PROGRAM GEMMA
VAR
	STEP_A6: INT := 0;
	DELAY_EJECTION_CARRIERS: TON;
	EJECT_CARRIERS: BOOL;
	F2_END: BOOL;
	STEP: STRING(20);
END_VAR

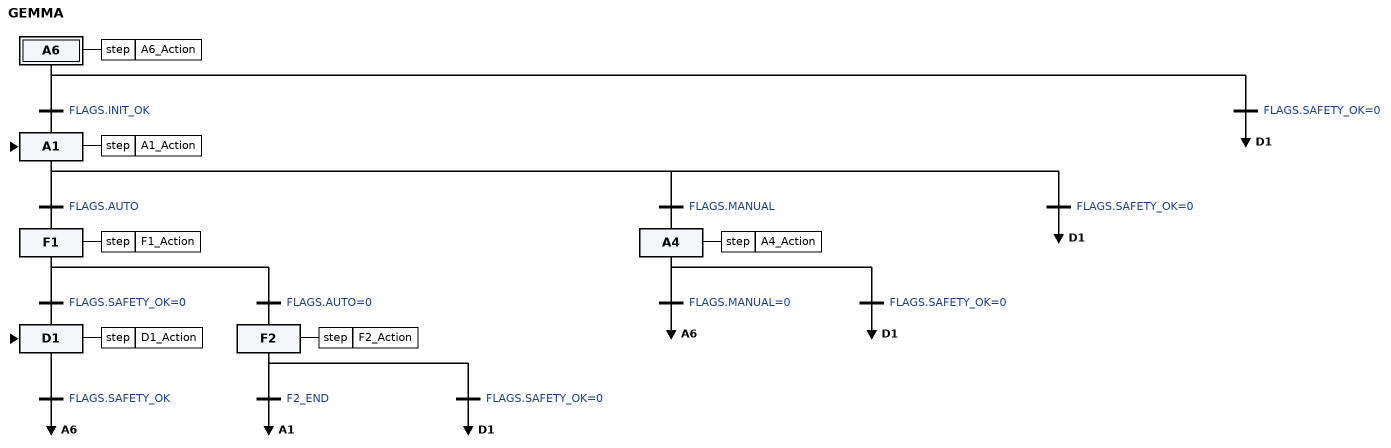
INITIAL_STEP A6_:  // name as stored: A6 
    A6_Action(N);  // step action
END_STEP
TRANSITION FROM A6_ TO A1
    := FLAGS.INIT_OK;
END_TRANSITION
TRANSITION FROM A6_ TO D1
    := FLAGS.SAFETY_OK=0;
END_TRANSITION
STEP A1:
    A1_Action(N);  // step action
END_STEP
TRANSITION FROM A1 TO F1
    := FLAGS.AUTO;
END_TRANSITION
TRANSITION FROM A1 TO A4
    := FLAGS.MANUAL;
END_TRANSITION
STEP A4:
    A4_Action(N);  // step action
END_STEP
TRANSITION FROM A4 TO A6
    := FLAGS.MANUAL=0;
END_TRANSITION
TRANSITION FROM A4 TO D1
    := FLAGS.SAFETY_OK=0;
END_TRANSITION
TRANSITION FROM A1 TO D1
    := FLAGS.SAFETY_OK=0;
END_TRANSITION
STEP F1:
    F1_Action(N);  // step action
END_STEP
TRANSITION FROM F1 TO D1
    := FLAGS.SAFETY_OK=0;
END_TRANSITION
TRANSITION FROM F1 TO F2
    := FLAGS.AUTO=0;
END_TRANSITION
STEP F2:
    F2_Action(N);  // step action
END_STEP
TRANSITION FROM F2 TO A1
    := F2_END;
END_TRANSITION
TRANSITION FROM F2 TO D1
    := FLAGS.SAFETY_OK=0;
END_TRANSITION
STEP D1:
    D1_Action(N);  // step action
END_STEP
TRANSITION FROM D1 TO A6
    := FLAGS.SAFETY_OK;
END_TRANSITION

ACTION F1_Action:
(*********************************************************
*
* F1
*
************************************************************)

STEP := 'F1';
END_ACTION

ACTION A6_Action:
(**************************************************************
*
*
* Initialisation
*
*
***************************************************************)
STEP:='A6';



CASE STEP_A6 OF

0: (*Init*)
	STEP_A6:=STEP_A6+1;

1: (*Initialise valves and variables*)

	GEN_1V1 				:=FALSE;	(*Vanne AIR*)
	GEN_CONVOYEUR			:=FALSE;	(*Relais convoyeur*)	
	
	ST1_1V1 	:=FALSE;		(*Vérin palette attente*)
	ST1_1V2 	:=FALSE;		(*Vérin palette bloquage*)
	ST1_1V3 	:=FALSE;		(*Vérin palette stop*)
	ST1_1V4 	:=FALSE;		(*Vérin connexion TOP*)
	ST1_1V5		:=FALSE;		(*Vérin connexion HT*)

	ST2_2V1 	:=FALSE;		(*Vérin palette attente*)
	ST2_2V2 	:=FALSE;		(*Vérin palette bloquage*)
	ST2_2V3 	:=FALSE;		(*Vérin palette stop*)
	ST2_2V4 	:=FALSE;		(*Vérin Hydro TOP*)
	ST2_2V5		:=FALSE;		(*Vérin hydro BOTTOM*)
	ST2_2V6		:=FALSE;		(*Vérin électrique*)
	ST2_2V7		:=FALSE;		(*Vérin by-pass*)
	
	ST2_POWER	:=FALSE;		(*Alimentation électrique pompe*)
	
	ST3_3V1 	:=FALSE;		(*Vérin palette attente*)
	ST3_3V2 	:=FALSE;		(*Vérin palette bloquage*)
	ST3_3V3 	:=FALSE;		(*Vérin palette stop*)
	ST3_3V4 	:=FALSE;		(*Vérin Hydro TOP*)
	ST3_3V5		:=FALSE;		(*Vérin hydro BOTTOM*)
	ST3_3V7		:=FALSE;		(*Vérin by-pass*)
	
	ST3_3V10 	:=FALSE;		(*Vanne avant la pompe*)
	ST3_3V11 	:=FALSE;		(*Vanne après la pompe*)
	ST3_3V12 	:=FALSE;		(*Vanne de blocage d'air pour le DELTA*)
	
	ST4_4V1 	:=FALSE;		(*Vérin palette attente*)
	ST4_4V2 	:=FALSE;		(*Vérin palette bloquage*)
	ST4_4V3 	:=FALSE;		(*Vérin palette stop*)
	ST4_4V4 	:=FALSE;		(*Vérin Hydro TOP*)
	ST4_4V5		:=FALSE;		(*Vérin hydro BOTTOM*)
	ST4_4V6		:=FALSE;		(*Vérin électrique*)
	ST4_4V7		:=FALSE;		(*Vérin by-pass*)
	
	ST4_4V10	:=FALSE;		(*Vanne avant la pompe*)
	ST4_4V12	:=FALSE;		(*Vanne après la vanne pilotée*)
	ST4_4V13	:=FALSE;		(*Vanne max flow*)

	ST4_POWER	:=FALSE;		(*Alimentation électrique pompe*)
	ST4_VIDANGE	:=FALSE;		(*Vidange balance*)
	
	ST5_5V1 	:=FALSE;		(*Vérin palette attente*)
	ST5_5V2 	:=FALSE;		(*Vérin palette bloquage*)
	ST5_5V3 	:=FALSE;		(*Vérin palette stop*)
	ST5_5V4 	:=FALSE;		(*Vérin Hydro TOP*)
	ST5_5V5		:=FALSE;		(*Vérin hydro BOTTOM*)
	ST5_5V6		:=FALSE;		(*Vérin électrique*)
	
	ST5_5V10	:=FALSE;		(*Vanne avant la pompe*)
	ST5_5V12	:=FALSE;		(*Vanne après la vanne pilotée*)
	ST5_5V13	:=FALSE;		(*Vanne max flow*)
	
	ST5_5V14	:=FALSE;		(*Vanne vidange vers égouts ou réservoir*)
	ST5_5V15	:=FALSE;			(*Vanne avant la pompe*)
	ST5_5V16	:=FALSE;		(*Vanne provenance eau du réservoir ou du déminéralisateur*)
	
	ST5_POWER	:=FALSE;		(*Alimentation électrique pompe*)
	ST5_VIDANGE	:=FALSE;		(*Vidange balance*)
	
	ST6_6V1 	:=FALSE;		(*Vérin palette attente*)
	ST6_6V2 	:=FALSE;		(*Vérin palette bloquage*)
	ST6_6V3 	:=FALSE;		(*Vérin palette stop*)
	ST6_6V4 	:=FALSE;		(*Vérin Hydro TOP*)
	ST6_6V5		:=FALSE;		(*Vérin hydro BOTTOM*)
	ST6_6V6		:=FALSE;		(*Vérin électrique*)
	ST6_6V7		:=FALSE;		(*Vérin by-pass*)
	
	ST6_6V10	:=FALSE;		(*Vanne avant la pompe*)
	ST6_6V11	:=FALSE;		(*Vanne après la pompe*)
	
	ST6_POWER	:=FALSE;		(*Alimentation électrique pompe*)
	
	ST7_7V1 	:=FALSE;		(*Vérin palette attente*)
	ST7_7V2 	:=FALSE;		(*Vérin palette bloquage*)
	ST7_7V3 	:=FALSE;		(*Vérin palette stop*)
	ST7_7V4 	:=FALSE;		(*Vérin Hydro TOP*)
	ST7_7V5		:=FALSE;		(*Vérin hydro BOTTOM*)
	ST7_7V6		:=FALSE;		(*Vérin électrique*)
	ST7_7V7		:=FALSE;		(*Vérin by-pass*)
	
	ST7_7V10	:=FALSE;		(*Vanne avant la pompe*)
	
	ST7_POWER	:=FALSE;		(*Alimentation électrique pompe*)
	
	ST8_8V1 	:=FALSE;		(*Vérin palette attente*)
	ST8_8V2 	:=FALSE;		(*Vérin palette bloquage*)
	ST8_8V3 	:=FALSE;		(*Vérin palette stop*)
	ST8_8V4 	:=FALSE;		(*Reserve*)
	
	ST9_9V1 	:=FALSE;		(*Vérin palette attente*)
	ST9_9V2 	:=FALSE;		(*Vérin palette bloquage*)
	ST9_9V3 	:=FALSE;		(*Vérin palette stop*)
	ST9_9V4 	:=FALSE;		(*Vérin rodless guide*)
	ST9_9V5 	:=FALSE;		(*Vérin slide table*)
	ST9_9V6 	:=FALSE;		(*Vérin gripper*)
	ST9_9V7 	:=FALSE;		(*Vérin liberateur electrique*)
	
	ST10_10V1 	:=TRUE;		(*Opérateur 1 - Vérin carrier stop*)
	ST10_10V2 	:=TRUE;		(*Opérateur 2 - Vérin carrier stop*)


	STEP_A6:=STEP_A6+1;

2: (*Start AIR and wait for ejection of all carriers on the conveyor*)

	GEN_1V1 := TRUE;
	GEN_CONVOYEUR := TRUE;
	EJECT_CARRIERS:=TRUE;

	STEP_A6:=STEP_A6+1;

3: (* Wait carriers ejection *)

	IF DELAY_EJECTION_CARRIERS.Q THEN
		EJECT_CARRIERS:=FALSE;
		STEP_A6:=STEP_A6+1;
	END_IF;
4: (*End of init *)

	FLAGS.INIT_OK:=TRUE;


ELSE
    ;
END_CASE;

(* FBs *)
DELAY_EJECTION_CARRIERS(IN:=EJECT_CARRIERS , PT:= DELAY_EJECT_CARRIERS);
END_ACTION

ACTION A1_Action:
(***************************************************************************
*
* A1
*
****************************************************************************)
STEP := 'A1';
END_ACTION

ACTION A4_Action:
STEP:= 'A4';
END_ACTION

ACTION D1_Action:
(*****************************************************************
*
* NOT AUS state
*
******************************************************************)

	STEP := 'D1';
	
	STEP_A6:=0;
	F2_END:=FALSE;

	FLAGS.INIT_OK			:=FALSE;
	FLAGS.MOTOR_Q1_INIT_OK	:=FALSE;
	FLAGS.AUTO				:=FALSE;
	FLAGS.MANUAL			:=FALSE;

	GEN_1V1 				:=FALSE;	(*Vanne AIR*)
	GEN_CONVOYEUR			:=FALSE;	(*Relais convoyeur*)	
	
	ST1_1V1 	:=FALSE;		(*Vérin palette attente*)
	ST1_1V2 	:=FALSE;		(*Vérin palette bloquage*)
	ST1_1V3 	:=FALSE;		(*Vérin palette stop*)
	ST1_1V4 	:=FALSE;		(*Vérin connexion TOP*)
	ST1_1V5		:=FALSE;		(*Vérin connexion HT*)

	ST2_2V1 	:=FALSE;		(*Vérin palette attente*)
	ST2_2V2 	:=FALSE;		(*Vérin palette bloquage*)
	ST2_2V3 	:=FALSE;		(*Vérin palette stop*)
	ST2_2V4 	:=FALSE;		(*Vérin Hydro TOP*)
	ST2_2V5		:=FALSE;		(*Vérin hydro BOTTOM*)
	ST2_2V6		:=FALSE;		(*Vérin électrique*)
	ST2_2V7		:=FALSE;		(*Vérin by-pass*)
	
	ST2_POWER	:=FALSE;		(*Alimentation électrique pompe*)
	
	ST3_3V1 	:=FALSE;		(*Vérin palette attente*)
	ST3_3V2 	:=FALSE;		(*Vérin palette bloquage*)
	ST3_3V3 	:=FALSE;		(*Vérin palette stop*)
	ST3_3V4 	:=FALSE;		(*Vérin Hydro TOP*)
	ST3_3V5		:=FALSE;		(*Vérin hydro BOTTOM*)
	ST3_3V7		:=FALSE;		(*Vérin by-pass*)
	
	ST3_3V10 	:=FALSE;		(*Vanne avant la pompe*)
	ST3_3V11 	:=FALSE;		(*Vanne après la pompe*)
	ST3_3V12 	:=FALSE;		(*Vanne de blocage d'air pour le DELTA*)
	
	ST4_4V1 	:=FALSE;		(*Vérin palette attente*)
	ST4_4V2 	:=FALSE;		(*Vérin palette bloquage*)
	ST4_4V3 	:=FALSE;		(*Vérin palette stop*)
	ST4_4V4 	:=FALSE;		(*Vérin Hydro TOP*)
	ST4_4V5		:=FALSE;		(*Vérin hydro BOTTOM*)
	ST4_4V6		:=FALSE;		(*Vérin électrique*)
	ST4_4V7		:=FALSE;		(*Vérin by-pass*)
	
	ST4_4V10	:=FALSE;		(*Vanne avant la pompe*)
	ST4_4V12	:=FALSE;		(*Vanne après la vanne pilotée*)
	ST4_4V13	:=FALSE;		(*Vanne max flow*)

	ST4_POWER	:=FALSE;		(*Alimentation électrique pompe*)
	ST4_VIDANGE	:=FALSE;		(*Vidange balance*)
	
	ST5_5V1 	:=FALSE;		(*Vérin palette attente*)
	ST5_5V2 	:=FALSE;		(*Vérin palette bloquage*)
	ST5_5V3 	:=FALSE;		(*Vérin palette stop*)
	ST5_5V4 	:=FALSE;		(*Vérin Hydro TOP*)
	ST5_5V5		:=FALSE;		(*Vérin hydro BOTTOM*)
	ST5_5V6		:=FALSE;		(*Vérin électrique*)
	
	ST5_5V10	:=FALSE;		(*Vanne avant la pompe*)
	ST5_5V12	:=FALSE;		(*Vanne après la vanne pilotée*)
	ST5_5V13	:=FALSE;		(*Vanne max flow*)
	
	ST5_5V14	:=FALSE;		(*Vanne vidange vers égouts ou réservoir*)
	ST5_5V15	:=FALSE;			(*Vanne avant la pompe*)
	ST5_5V16	:=FALSE;		(*Vanne provenance eau du réservoir ou du déminéralisateur*)
	
	ST5_POWER	:=FALSE;		(*Alimentation électrique pompe*)
	ST5_VIDANGE	:=FALSE;		(*Vidange balance*)
	
	ST6_6V1 	:=FALSE;		(*Vérin palette attente*)
	ST6_6V2 	:=FALSE;		(*Vérin palette bloquage*)
	ST6_6V3 	:=FALSE;		(*Vérin palette stop*)
	ST6_6V4 	:=FALSE;		(*Vérin Hydro TOP*)
	ST6_6V5		:=FALSE;		(*Vérin hydro BOTTOM*)
	ST6_6V6		:=FALSE;		(*Vérin électrique*)
	ST6_6V7		:=FALSE;		(*Vérin by-pass*)
	
	ST6_6V10	:=FALSE;		(*Vanne avant la pompe*)
	ST6_6V11	:=FALSE;		(*Vanne après la pompe*)
	
	ST6_POWER	:=FALSE;		(*Alimentation électrique pompe*)
	
	ST7_7V1 	:=FALSE;		(*Vérin palette attente*)
	ST7_7V2 	:=FALSE;		(*Vérin palette bloquage*)
	ST7_7V3 	:=FALSE;		(*Vérin palette stop*)
	ST7_7V4 	:=FALSE;		(*Vérin Hydro TOP*)
	ST7_7V5		:=FALSE;		(*Vérin hydro BOTTOM*)
	ST7_7V6		:=FALSE;		(*Vérin électrique*)
	ST7_7V7		:=FALSE;		(*Vérin by-pass*)
	
	ST7_7V10	:=FALSE;		(*Vanne avant la pompe*)
	
	ST7_POWER	:=FALSE;		(*Alimentation électrique pompe*)
	
	ST8_8V1 	:=FALSE;		(*Vérin palette attente*)
	ST8_8V2 	:=FALSE;		(*Vérin palette bloquage*)
	ST8_8V3 	:=FALSE;		(*Vérin palette stop*)
	ST8_8V4 	:=FALSE;		(*Reserve*)
	
	ST9_9V1 	:=FALSE;		(*Vérin palette attente*)
	ST9_9V2 	:=FALSE;		(*Vérin palette bloquage*)
	ST9_9V3 	:=FALSE;		(*Vérin palette stop*)
	ST9_9V4 	:=FALSE;		(*Vérin rodless guide*)
	ST9_9V5 	:=FALSE;		(*Vérin slide table*)
	ST9_9V6 	:=FALSE;		(*Vérin gripper*)
	ST9_9V7 	:=FALSE;		(*Vérin liberateur electrique*)
	
	ST10_10V1 	:=FALSE;		(*Opérateur 1 - Vérin carrier stop*)
	ST10_10V2 	:=FALSE;		(*Opérateur 2 - Vérin carrier stop*)
END_ACTION

ACTION F2_Action:
STEP := 'F2';
END_ACTION

END_PROGRAM

(* stored: Version 1.1.0.1, ProductVersion 3.1.0.26
   POU GEMMA: Id {caba80c3-9027-4275-b033-341dad53175a}
   Action F1_Action: Id {263b9e56-4c1a-486a-b55d-67d5b96b5874}
   Action A6_Action: Id {35d361ca-ae43-4b85-80cd-dcdb3546dd6b}
   Action A1_Action: Id {9028462a-cc66-4cee-b37e-215f3831f50c}
   Action A4_Action: Id {9cd56dcb-5c8e-47aa-8797-cf3b6f27d093}
   Action D1_Action: Id {b6d83183-e2ee-4c3f-a3f5-f6e80eed41a1}
   Action F2_Action: Id {e2a6bd08-06eb-486c-9ebb-86878540e224} *)
